{attribute 'GeneratedUsingTerminal: EP6224-0002-0016'}
{attribute addProperty BoxType "EP6224-0002-0016"}
{attribute addProperty Id "DeviceState_Inputs_DeviceDeviceState_Inputs_Device_A12105982"}
{attribute addProperty CRC "1394749468"}
{attribute addProperty Size "2"}
TYPE Module_1_DeviceState_Inputs_Device_5322301C :
STRUCT
	{attribute addProperty Name "DeviceState_Inputs_Device"}
	DeviceState_Inputs_Device  : DeviceState_Inputs_Device_A1210598;
END_STRUCT
END_TYPE

(* stored: Version 1.2.0.0, ProductVersion 3.1.4024.9
   DUT Module_1_DeviceState_Inputs_Device_5322301C: Id {91bce881-40b3-4dc4-94bb-6a94b3e9e11f} *)
